TYPE T_NewRFID_DtChn :
STRUCT
	// new RF ID
	strID: STRING;			// configurable if Tag or Tray ID
	uliTagID: ULINT;
	dtTimestamp: DT;
	intDataState: INT;	
END_STRUCT
END_TYPE

(* stored: Version 1.1.0.1, ProductVersion 3.1.0.20
   DUT T_NewRFID_DtChn: Id {8f51bc39-bcf8-4bc4-978c-c474f1fb6d1b} *)
